TEXTLIST ManualText
  0 = ' \n  取料Y轴\n1:初始位 2:Line0取料位 3:Line1取料位 4:Line3取料位\n\n   取料Z轴\n1:上升位 2:下降位_Line0 3:下降位_Line1\n\n   下UC_Y轴\n1:初始位 2:Line2取料位 3:Line3取料位 4:下UC位\n' | Chinese: ' \n  取料Y轴\n1:初始位 2:Line0取料位 3:Line1取料位 4:Line3取料位\n\n   取料Z轴\n1:上升位 2:下降位_Line0 3:下降位_Line1\n\n   下UC_Y轴\n1:初始位 2:Line2取料位 3:Line3取料位 4:下UC位\n' | English: ' \nPick the y axis\nThe initial bit is the initial bit 2:line0\n\nPick the z axis\nDrop _line0 3: drop _line1\n\nThe lower uc_y axis\n1: the initial bit 2:line2 takes the material bit \n3:line3 takes the material bit 4: the lower uc bit' | Vietnamese: ' \nLấy vật liệu trên trục Y\n1: ban đầu bit 2: dòng 0 cấp 3: dòng 1 cấp 4: dòng 3 cấp\n\nLấy trục Z\n1: nâng lên 2: hạ xuống bit _dòng 0 3: hạ xuống bit _dòng 1\n\nTrục dưới UC_Y\n1: bắt đầu bit 2: dòng 2 cấp 3: dòng 3 cấp 4: UC'
  1 = '   \n 流线1和流线3上料站:\n     顶升气缸缩回时,旋转气缸不动作.\n 流线2和流线3解锁站:\n     解锁侧推气缸2伸出时,解锁旋转气缸不缩回.\n     解锁侧推气缸2伸出时,下UC升降气缸不动作.\n     下UC旋转气缸伸出时,下UC升降气缸不动作.\n     下UC升降气缸缩回时,下UC旋转气缸不动作.\n RH311和LH311:\n     取料模组升降气缸1伸出时,取料Y轴不动作.\n     下UC模组升降气缸伸出时,下UC_Y轴不动作.\n     下UC模组摆动气缸伸出时,下UC_Y轴不动作.\n RH367和LH367:\n     取料模组升降气缸1伸出且升降气缸2伸出,\n 取料Y轴不动作.'
   = ''
END_TEXTLIST

(* stored: Version 1.1.0.1, ProductVersion 3.1.4024.3
   TextList ManualText: Id {3ad67886-0b61-436a-ac96-59136b45e612} *)
